TYPE DUT_MotionStage :
STRUCT
	// Hardware
	Axis: AXIS_REF;
	bLimFwd AT %I*: BOOL;
	bLimBwd AT %I*: BOOL;
	bHome AT %I*: BOOL;
	bBrake AT %Q*: BOOL;
	bSTO AT %I*: BOOL;
	
	// Psuedo-hardware
	bLimAllFwd: BOOL:=FALSE; // Forward enable EPS summary
	bLimAllBwd: BOOL:=FALSE; // Forward enable EPS summary 
	
	bLimGntFwd: BOOL:=FALSE; // Forward virtual gantry limit switch
	bLimGntBwd: BOOL:=FALSE; // Reverse virtual gantry limit switch
	
	// Settings
	bPowerSelf: BOOL:=TRUE;
	nEnableMode: INT:=ENUM_StageEnableMode.STAGE_ENABLE_MOTION;
	nBrakeMode: INT:=ENUM_StageBrakeMode.STAGE_BRAKE_DISABLED;
	nHomingMode: INT:=ENUM_EpicsHomeCmd.EPICS_MOTOR_HOME_NONE;
	
	bGantryAxis: BOOL:=FALSE; // Set true to activate gantry EPS
	fGantryTol: LREAL:=0; // Set to gantry difference tolerance
	nEncRef: ULINT:=0; // Encoder count at which this axis is aligned with other axis
	
	// Commands
	bEnable: BOOL;
	bReset: BOOL;
	bExecute: BOOL;
	
	// Args
	nCommand: INT;
	nCmdData: INT;
	fPosition: LREAL;
	fVelocity: LREAL;
	fAcceleration: LREAL;
	fDeceleration: LREAL;
	fHomePosition: LREAL;
	
	// Info
	nMotionAxisID: UDINT:=0;
	
	// Returns
	bEnabled: BOOL;
	bBusy: BOOL;
	bDone: BOOL;
	bError: BOOL;
	sErrorMessage: STRING;
	stAxisStatus: DUT_AxisStatus_v0_01;
END_STRUCT
END_TYPE

(* stored: Version 1.1.0.1, ProductVersion 3.1.4020.14
   DUT DUT_MotionStage: Id {10b5775d-5646-4d55-ad77-40abc3888de3} *)
